FUNCTION_BLOCK FB_JoystickInputScaling
// LREAL: Long Real decimal number
// INT: [-32768, 32767]	
// BOOL: True/False

// Input variables
VAR_INPUT
	bEnable 				: BOOL;
	nRawInput 				: INT;
	fMaxValue 				: LREAL;
	fMaxInputValue			: LREAL;
	fMinInputValue 			: LREAL;
	fNeutralInputValue  	: LREAL;
	fNeutralDeadband		: LREAL;
END_VAR

// Output variables
VAR_OUTPUT
	fOutput : LREAL;
END_VAR

// Variables
VAR
	fRawInput : LREAL;
	fTempInput : LREAL; // Temporary input
	fTempOutput : LREAL; // Temporary output

	fMaxOutputValue  		: LREAL := 1.0;
	fMinOutputValue  		: LREAL := -1.0;
	fNeutralOutputValue  	: LREAL := 0.0;
END_VAR

// Crane is only supported for movement in the y-axis (up/down)

fRawInput := INT_TO_LREAL(nRawInput); // Converts input to decimal number
fTempInput := fRawInput - fNeutralInputValue; // Defines joystick neutral point 

IF fTempInput > fNeutralDeadband THEN // Checks if joystick is moved above the neutral deadband (positive y) 
	fTempOutput := fTempInput/(fMaxInputValue - fNeutralInputValue); // Scales positive movement [0,1]
ELSIF fTempInput < -fNeutralDeadband THEN // Checks if joystick is moved below the neutral deadband (negative y)
	fTempOutput := fTempInput/(fNeutralInputValue - fMinInputValue); // Scales negative movement [-1,0]
ELSE
	fTempOutput := 0.0; // If joystick is inside deadzone, fTempOutput = 0
END_IF

IF NOT(bEnable) THEN // If bEnable is not true, set fOutput = 0
	fOutput := 0.0;
ELSE
	fOutput := LIMIT(fMinOutputValue * fMaxValue, fTempOutput * fMaxValue, fMaxOutputValue* fMaxValue); 
	// Calculates output signal within safety limits (Min, Output, Max)
END_IF

END_FUNCTION_BLOCK

(* stored: Version 1.1.0.1
   POU FB_JoystickInputScaling: Id {45abe8f1-3862-4b14-9ee2-cf88212f6af6}, SpecialFunc None *)
